FUNCTION Convert_BYTE_TO_LWORD : BOOL
VAR_INPUT
	in : BYTE;
	out : REFERENCE TO LWORD;
END_VAR
VAR
	converted : LWORD;
END_VAR

converted := BYTE_TO_LWORD(in);

IF (LWORD_TO_BYTE(converted) <> in) THEN
	RETURN;
END_IF

out := converted;
Convert_BYTE_TO_LWORD := TRUE;

END_FUNCTION

(* stored: Version 1.1.0.1, ProductVersion 3.1.4024.12
   POU Convert_BYTE_TO_LWORD: Id {1a4d5ea9-bacd-40d0-aaf5-a1f1abe5d617}, SpecialFunc None *)
